(* CoDeSys 2.3 export: BUTTON.EXP *)

(* POU Components/Button, ST *)
FUNCTION_BLOCK Button
VAR_INPUT
	input: BOOL;
END_VAR

VAR
	EdgeDetection:EdgeDetection := (onFallingEdge:=1);
	fallingEdge:BOOL;
	longPressed:BOOL;
	timer:Delay:= (timeSetup:= 20);
	tmp:BOOL;
END_VAR
EdgeDetection(input:=input, output => tmp);
fallingEdge := tmp AND NOT timer.afterTime;

timer(start:= input);
longPressed:= timer.afterTimeImpulse;
END_FUNCTION_BLOCK
